{attribute 'GeneratedUsingTerminal: EK1100-0000-0018'}
{attribute addProperty BoxType "EK1100-0000-0018"}
{attribute addProperty Id "Beckhoff_ER3xxxEK1122Beckhoff_ER3xxxEK1122_48B49356618"}
{attribute addProperty CRC "1612479836"}
{attribute addProperty Size "618"}
TYPE Beckhoff_ER3xxx_601C7D5C EXTENDS EK1100_AB5A9467 :
STRUCT
	{attribute addProperty Name "Beckhoff_ER3xxxEK1122"}
	{attribute addProperty PreviousPort "Beckhoff ER3xxx : B"}
	Beckhoff_ER3xxxEK1122 : Beckhoff_ER3xxxEK1122_48B49356;
END_STRUCT
END_TYPE

(* stored: Version 1.2.0.0, ProductVersion 3.1.4024.9
   DUT Beckhoff_ER3xxx_601C7D5C: Id {57fee5de-9114-4a83-917a-274a155cb57b} *)
